PROGRAM MAIN
VAR
END_VAR

Control_FBD();

END_PROGRAM

(* stored: Version 1.1.0.1, ProductVersion 3.1.4022.12
   POU MAIN: Id {08a3c80a-9d54-4bd3-a860-80de0df9675b}, SpecialFunc None *)
